// TIA Portal V19 export
TYPE "udt_RollformingMng_Target"
   STRUCT
      Ready : Bool;
      P_ID : DInt;
      O_ID : DInt;
      Beam_Code : Int;
      X_Start : LReal;
      X_End : LReal;
      TargetTolerance : LReal;
      PartLength : LReal;
      DrawHead : Bool;
      MarkHead : Bool;
      WeldPresence : Bool;
   END_STRUCT;
END_TYPE
